// TIA Portal V17 export
// export: Created 2025-03-07T09:19:56.4658Z, ExportSetting WithDefaults, DisplayName Totally Integrated Automation Portal, DisplayVersion V17 Update 8, DisplayName TIA Portal Openness, DisplayVersion V17 Update 8, DisplayName TIA Portal Version Control Interface, DisplayVersion V17, DisplayName SINAMICS Startdrive Advanced, DisplayVersion V17 SP2, DisplayName SINAMICS Startdrive G110M, G120, G120C, G120D, G120P, G115D, DisplayVersion V17 SP2, DisplayName SINAMICS Startdrive G130, G150, S120, S150, SINAMICS MV, S210, DisplayVersion V17 SP2, DisplayName STEP 7 Professional, DisplayVersion V17 Update 8, DisplayName SINUMERIK ONE STEP 7 Toolbox, DisplayVersion V17 Update 12, DisplayName SINUMERIK 840D sl STEP 7 Toolbox, DisplayVersion V17 Update 12, DisplayName STEP 7 Safety, DisplayVersion V17 Update 6, DisplayName WinCC Advanced, DisplayVersion V17 Update 8
TYPE "ROBOT_TOOL_STATUS"
// stored: IsFailsafeCompliant false
   STRUCT
      EMPTY : Bool;   // ROBOT TOOL GRIPPER EMPTY
      ANY_PART_PRESENT : Bool;   // ROBOT TOOL GRIPPER ANY PART PRESENT
      ALL_PARTS_PRESENT : Bool;   // ROBOT TOOL GRIPPER ALL PARTS PRESENT
      SPARE_0_3 : Bool;
      SPARE_0_4 : Bool;
      SPARE_0_5 : Bool;
      SPARE_0_6 : Bool;
      SPARE_0_7 : Bool;
      PART_A_PRESENT_INPUT : Bool;   // PART A PRESENT INPUT
      PART_B_PRESENT_INPUT : Bool;   // PART B PRESENT_INPUT
      PART_C_PRESENT_INPUT : Bool;   // PART C PRESENT INPUT
      PART_D_PRESENT_INPUT : Bool;   // PART D PRESENT INPUT
      PART_E_PRESENT_INPUT : Bool;   // PART E PRESENT INPUT
      SPARE_1_5 : Bool;
      SPARE_1_6 : Bool;
      SPARE_1_7 : Bool;
      DISCORDANCY_PART_A : Bool;   // DISCORDANCY PART A
      DISCORDANCY_PART_B : Bool;   // DISCORDANCY PART B
      DISCORDANCY_PART_C : Bool;   // DISCORDANCY PART C
      DISCORDANCY_PART_D : Bool;   // DISCORDANCY PART D
      DISCORDANCY_PART_E : Bool;   // DISCORDANCY PART E
      SPARE_2_5 : Bool;
      SPARE_2_6 : Bool;
      DISCORDANCY_FAULT : Bool;   // DISCORDANCY FAULT
      ANY_NEW_PART_PRESENT : Bool;   // ANY NEW PART PRESENT
      ALL_NEW_PARTS_PRESENT : Bool;   // ALL NEW PARTS PRESENT
      NEW_PART_A : Bool;
      NEW_PART_B : Bool;
      NEW_PART_C : Bool;
      NEW_PART_D : Bool;
      NEW_PART_E : Bool;
      SPARE_3_7 : Bool;
      ANY_FNSHD_PART_PRESENT_U1 : Bool;   // ANY FINISHED PART PRESENT FROM UNIT 1
      ALL_FNSHD_PART_PRESENT_U1 : Bool;   // ALL FINISHED PARTS PRESENT FROM UNIT 1
      FINISHED_FROM_U1_PA : Bool;   // PART FINISHED FROM UNIT 1 - PART "A"
      FINISHED_FROM_U1_PB : Bool;   // PART FINISHED FROM UNIT 1 - PART "B"
      FINISHED_FROM_U1_PC : Bool;   // PART FINISHED FROM UNIT 1 - PART "C"
      FINISHED_FROM_U1_PD : Bool;   // PART FINISHED FROM UNIT 1 - PART "D"
      FINISHED_FROM_U1_PE : Bool;   // PART FINISHED FROM UNIT 1 - PART "E"
      SPARE_4_7 : Bool;
      ANY_FNSHD_PART_PRESENT_U2 : Bool;   // ANY FINISHED PART PRESENT FROM UNIT 2
      ALL_FNSHD_PART_PRESENT_U2 : Bool;   // ALL FINISHED PARTS PRESENT FROM UNIT 2
      FINISHED_FROM_U2_PA : Bool;   // PART FINISHED FROM UNIT 2 - PART "A"
      FINISHED_FROM_U2_PB : Bool;   // PART FINISHED FROM UNIT 2 - PART "B"
      FINISHED_FROM_U2_PC : Bool;   // PART FINISHED FROM UNIT 2 - PART "C"
      FINISHED_FROM_U2_PD : Bool;   // PART FINISHED FROM UNIT 2 - PART "D"
      FINISHED_FROM_U2_PE : Bool;   // PART FINISHED FROM UNIT 2 - PART "E"
      SPARE_5_7 : Bool;
      SPARE_6_0 : Byte;
      SPARE_7_0 : Byte;
      SPARE_8_0 : Byte;
      SPARE_9_0 : Byte;
      ANY_PART_REJECTED_U1 : Bool;   // ANY PART REJECTED FROM UNIT 1
      ALL_PARTS_REJTD_PRESENT_U1 : Bool;   // ALL PARTS REJECTED FROM UNIT 1
      REJECTED_FROM_U1_PA : Bool;   // REJECTED FROM UNIT 1 - PART "A"
      REJECTED_FROM_U1_PB : Bool;   // REJECTED FROM UNIT 1 - PART "B"
      REJECTED_FROM_U1_PC : Bool;   // REJECTED FROM UNIT 1 - PART "C"
      REJECTED_FROM_U1_PD : Bool;   // REJECTED FROM UNIT 1 - PART "D"
      REJECTED_FROM_U1_PE : Bool;   // REJECTED FROM UNIT 1 - PART "E"
      SPARE_10_5 : Bool;
      ANY_PART_REJECTED_U2 : Bool;   // ANY PART REJECTED FROM UNIT 2
      ALL_PARTS_REJTD_PRESENT_U2 : Bool;   // ALL PARTS REJECTED FROM UNIT 2
      REJECTED_FROM_U2_PA : Bool;   // REJECTED FROM UNIT 2 - PART "A"
      REJECTED_FROM_U2_PB : Bool;   // REJECTED FROM UNIT 2 - PART "B"
      REJECTED_FROM_U2_PC : Bool;   // REJECTED FROM UNIT 2 - PART "C"
      REJECTED_FROM_U2_PD : Bool;   // REJECTED FROM UNIT 2 - PART "D"
      REJECTED_FROM_U2_PE : Bool;   // REJECTED FROM UNIT 2 - PART "E"
      SPARE_11_5 : Bool;
      SPARE_11_6 : Bool;
      SPARE_11_7 : Bool;
      SPARE_12_0 : Byte;
      SPARE_13_0 : Byte;
      ANY_QC_PART_U1_PA : Bool;   // ANY PART TO QUALITY CHECK FROM UNIT 1
      ALL_QC_PART_U1_PA : Bool;   // ALL PARTS TO QUALITY CHECK FROM UNIT 1
      QC_FROM_U1_PA : Bool;   // QUALITY CHECK FROM UNIT 1 - PART "A"
      QC_FROM_U1_PB : Bool;   // QUALITY CHECK FROM UNIT 1 - PART "B"
      QC_FROM_U1_PC : Bool;   // QUALITY CHECK FROM UNIT 1 - PART "C"
      QC_FROM_U1_PD : Bool;   // QUALITY CHECK FROM UNIT 1 - PART "D"
      QC_FROM_U1_PE : Bool;   // QUALITY CHECK FROM UNIT 1 - PART "E"
      SPARE_14_7 : Bool;
      ANY_QC_PART_U2_PA : Bool;   // ANY PART TO QUALITY CHECK FROM UNIT 2
      ALL_QC_PART_U2_PA : Bool;   // ALL PARTS TO QUALITY CHECK FROM UNIT 2
      QC_FROM_U2_PA : Bool;   // QUALITY CHECK FROM UNIT 2 - PART "A"
      QC_FROM_U2_PB : Bool;   // QUALITY CHECK FROM UNIT 2 - PART "B"
      QC_FROM_U2_PC : Bool;   // QUALITY CHECK FROM UNIT 2 - PART "C"
      QC_FROM_U2_PD : Bool;   // QUALITY CHECK FROM UNIT 2 - PART "D"
      QC_FROM_U2_PE : Bool;   // QUALITY CHECK FROM UNIT 2 - PART "E"
      SPARE_15_7 : Bool;
      SPARE_16_0 : Byte;
      SPARE_17_0 : Byte;
      SPARE_18_0 : Byte;
      SPARE_19_0 : Byte;
   END_STRUCT;
END_TYPE
